// TwinCAT 3 PLC project carWash
// ProgramVersion: 3.1.4023.0
// libraries:
//   Tc2_Standard, * (Beckhoff Automation GmbH)
//   Tc2_System, * (Beckhoff Automation GmbH)
//   Tc3_Module, * (Beckhoff Automation GmbH)
// project tree:
//   / PlcTask.TcTTO
//   POUs/ MAIN.TcPOU
// real-time tasks:
//   TASK PlcTask: cycle T#10ms, priority 20, ADS port 350

CONFIGURATION carWash
    RESOURCE PLC ON TwinCAT3
        TASK PlcTask(INTERVAL := T#10ms, PRIORITY := 20);
        PROGRAM MAIN WITH PlcTask : MAIN;
    END_RESOURCE
END_CONFIGURATION

// ---- POUs/MAIN.TcPOU
PROGRAM MAIN
VAR
	preLavaggio : BOOL := FALSE;
	lavaggioInterno : BOOL := FALSE;
	sapone : BOOL := FALSE;
	risciacquo :BOOL := FALSE;
	posPreparazione :BOOL := FALSE;
	{attribute 'OPC.UA.DA' := '1'}
	polizia :BOOL := FALSE;
	postoAuto :BOOL := FALSE;
	postoMoto :BOOL := FALSE;
	start :BOOL := FALSE;
	reset :BOOL := FALSE;
	pause :BOOL := FALSE;
	moto :BOOL := FALSE;
	auto:BOOL := FALSE;
	fineProcessi :BOOL := FALSE;
	{attribute 'OPC.UA.DA' := '1'}
	costoAuto :INT := 0;
	{attribute 'OPC.UA.DA' := '1'}
	costoMoto :INT := 0;
	numeroStep :INT := 0;
	dx :BOOL := FALSE;
	sx :BOOL := FALSE;
	giu :BOOL := FALSE;
	allarme :BOOL := FALSE;
	
END_VAR

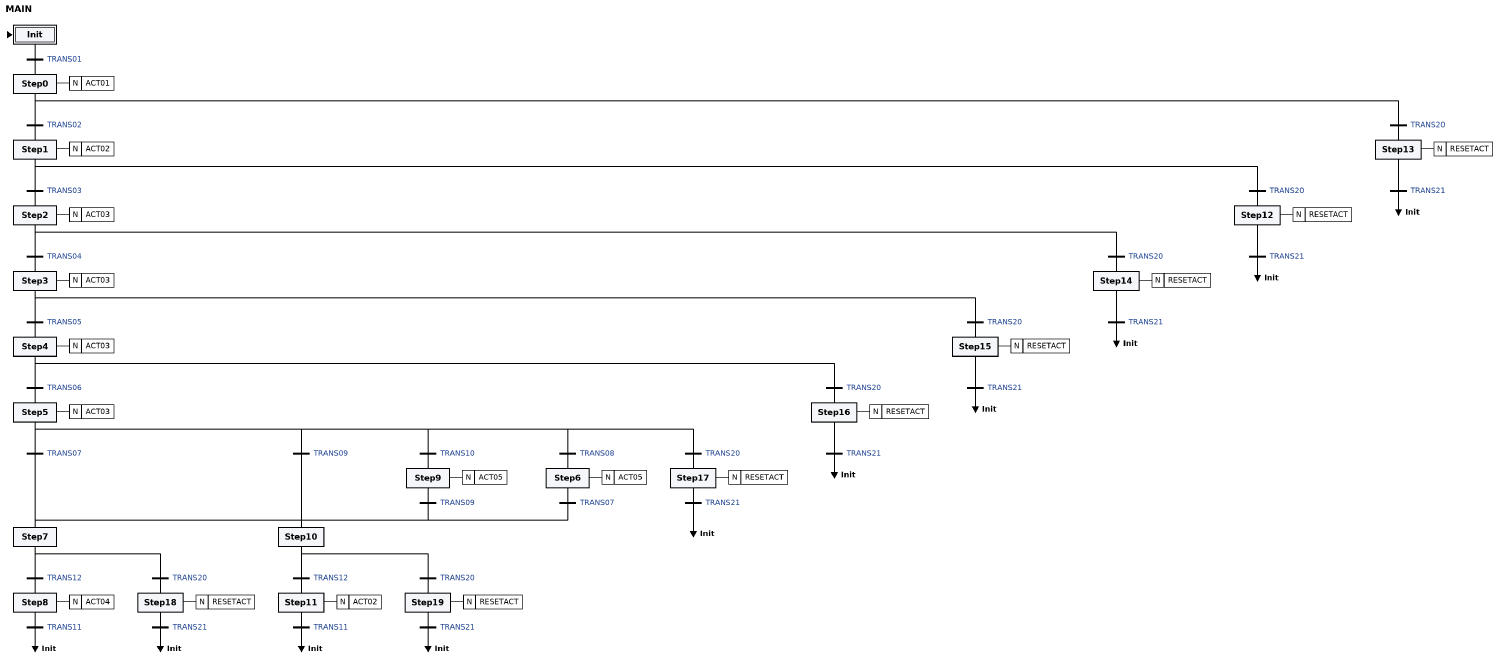
INITIAL_STEP Init:
END_STEP
TRANSITION FROM Init TO Step0
    := TRANS01;
END_TRANSITION
STEP Step0:
    ACT01(N);
END_STEP
TRANSITION FROM Step0 TO Step1
    := TRANS02;
END_TRANSITION
TRANSITION FROM Step0 TO Step13
    := TRANS20;
END_TRANSITION
STEP Step13:
    RESETACT(N);
END_STEP
TRANSITION FROM Step13 TO Init
    := TRANS21;
END_TRANSITION
STEP Step1:
    ACT02(N);
END_STEP
TRANSITION FROM Step1 TO Step2
    := TRANS03;
END_TRANSITION
TRANSITION FROM Step1 TO Step12
    := TRANS20;
END_TRANSITION
STEP Step12:
    RESETACT(N);
END_STEP
TRANSITION FROM Step12 TO Init
    := TRANS21;
END_TRANSITION
STEP Step2:
    ACT03(N);
END_STEP
TRANSITION FROM Step2 TO Step3
    := TRANS04;
END_TRANSITION
TRANSITION FROM Step2 TO Step14
    := TRANS20;
END_TRANSITION
STEP Step14:
    RESETACT(N);
END_STEP
TRANSITION FROM Step14 TO Init
    := TRANS21;
END_TRANSITION
STEP Step3:
    ACT03(N);
END_STEP
TRANSITION FROM Step3 TO Step4
    := TRANS05;
END_TRANSITION
TRANSITION FROM Step3 TO Step15
    := TRANS20;
END_TRANSITION
STEP Step15:
    RESETACT(N);
END_STEP
TRANSITION FROM Step15 TO Init
    := TRANS21;
END_TRANSITION
STEP Step4:
    ACT03(N);
END_STEP
TRANSITION FROM Step4 TO Step5
    := TRANS06;
END_TRANSITION
TRANSITION FROM Step4 TO Step16
    := TRANS20;
END_TRANSITION
STEP Step16:
    RESETACT(N);
END_STEP
TRANSITION FROM Step16 TO Init
    := TRANS21;
END_TRANSITION
STEP Step5:
    ACT03(N);
END_STEP
TRANSITION FROM Step5 TO Step7
    := TRANS07;
END_TRANSITION
TRANSITION FROM Step5 TO Step10
    := TRANS09;
END_TRANSITION
TRANSITION FROM Step5 TO Step9
    := TRANS10;
END_TRANSITION
STEP Step9:
    ACT05(N);
END_STEP
TRANSITION FROM Step9 TO Step10
    := TRANS09;
END_TRANSITION
STEP Step10:
END_STEP
TRANSITION FROM Step10 TO Step11
    := TRANS12;
END_TRANSITION
TRANSITION FROM Step10 TO Step19
    := TRANS20;
END_TRANSITION
STEP Step19:
    RESETACT(N);
END_STEP
TRANSITION FROM Step19 TO Init
    := TRANS21;
END_TRANSITION
STEP Step11:
    ACT02(N);
END_STEP
TRANSITION FROM Step11 TO Init
    := TRANS11;
END_TRANSITION
TRANSITION FROM Step5 TO Step6
    := TRANS08;
END_TRANSITION
STEP Step6:
    ACT05(N);
END_STEP
TRANSITION FROM Step6 TO Step7
    := TRANS07;
END_TRANSITION
TRANSITION FROM Step5 TO Step17
    := TRANS20;
END_TRANSITION
STEP Step17:
    RESETACT(N);
END_STEP
TRANSITION FROM Step17 TO Init
    := TRANS21;
END_TRANSITION
STEP Step7:
END_STEP
TRANSITION FROM Step7 TO Step8
    := TRANS12;
END_TRANSITION
TRANSITION FROM Step7 TO Step18
    := TRANS20;
END_TRANSITION
STEP Step18:
    RESETACT(N);
END_STEP
TRANSITION FROM Step18 TO Init
    := TRANS21;
END_TRANSITION
STEP Step8:
    ACT04(N);
END_STEP
TRANSITION FROM Step8 TO Init
    := TRANS11;
END_TRANSITION

ACTION ACT01:
start := FALSE;
END_ACTION

ACTION ACT02:
dx := TRUE;
END_ACTION

ACTION ACT03:
giu := TRUE;
dx := FALSE;
END_ACTION

ACTION ACT04:
sx := TRUE;
giu := FALSE;
polizia :=FALSE;
allarme := TRUE;
END_ACTION

ACTION ACT05:
polizia := TRUE;
END_ACTION

ACTION ACT06:
dx := TRUE;
giu := FALSE;
polizia :=FALSE;
allarme := TRUE;
END_ACTION

ACTION RESETACT:
	preLavaggio:= FALSE;
	lavaggioInterno := FALSE;
	sapone := FALSE;
	risciacquo  := FALSE;
	posPreparazione  := FALSE;
	polizia  := FALSE;
	postoAuto  := FALSE;
	postoMoto := FALSE;
	start  := FALSE;
	reset  := FALSE;
	pause  := FALSE;
	moto := FALSE;
	auto:= FALSE;
	fineProcessi := FALSE;
	costoAuto := 0;
	costoMoto := 0;
	numeroStep  := 0;
	dx := FALSE;
	sx  := FALSE;
	giu  := FALSE;
	allarme  := FALSE;
END_ACTION

TRANSITION TRANS01:
start;
END_TRANSITION

TRANSITION TRANS02:
(moto OR auto) and numeroStep=1;
END_TRANSITION

TRANSITION TRANS03:
numeroStep=2;
END_TRANSITION

TRANSITION TRANS04:
numeroStep=3;
END_TRANSITION

TRANSITION TRANS05:
numeroStep=4;
END_TRANSITION

TRANSITION TRANS06:
numeroStep=5;
END_TRANSITION

TRANSITION TRANS07:
numeroStep = 6 and costoMoto=5 and moto;
END_TRANSITION

TRANSITION TRANS08:
numeroStep=6 and costoMoto=0 AND moto;
END_TRANSITION

TRANSITION TRANS09:
numeroStep = 6 and costoAuto=10 and auto;
END_TRANSITION

TRANSITION TRANS10:
numeroStep=6 and costoAuto=0 AND auto;
END_TRANSITION

TRANSITION TRANS11:
numeroStep = 0 and (postoMoto=TRUE or postoAuto=TRUE);
END_TRANSITION

TRANSITION TRANS12:
numeroStep = 7;
END_TRANSITION

TRANSITION TRANS20:
RESET;
END_TRANSITION

TRANSITION TRANS21:
numeroStep = 0;
END_TRANSITION

END_PROGRAM
